FUNCTION_BLOCK CompareInts (* Basic FB with empty ECC *)
  (* Standard: 61499-2 *)
  (* Version 1.0, 2022-02-08, ki-do *)
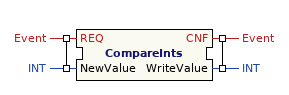
  EVENT_INPUT
    REQ WITH NewValue;
  END_EVENT
  EVENT_OUTPUT
    CNF WITH WriteValue;
  END_EVENT
  VAR_INPUT
    NewValue : INT;
  END_VAR
  VAR_OUTPUT
    WriteValue : INT;
  END_VAR
  VAR
    OldValue : INT := -32767; (* Internal Variable *)
  END_VAR
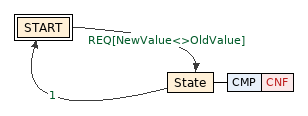
  EC_STATES
    START; (* Initial State *)
    State : CMP -> CNF;
  END_STATES
  EC_TRANSITIONS
    START TO State := REQ[NewValue<>OldValue];
    State TO START := 1;
  END_TRANSITIONS
  ALGORITHM CMP IN ST: (* New Algorithm *)
WriteValue:=NewValue;
OldValue:=NewValue;
  END_ALGORITHM
END_FUNCTION_BLOCK
